{attribute 'enable_dynamic_creation'}
FUNCTION_BLOCK Line EXTENDS Object IMPLEMENTS ILine
VAR_INPUT
END_VAR
VAR_OUTPUT
END_VAR
VAR
	content :STRING(255);
	number :LREAL;
END_VAR

(*

short summary
=================
This abstract property returns the class name of the concrete object, 
which is useful for logging/debugging purpose or to check the class name
for ``__DELETE`` in factories (sometimes it's necessary to do more 
than just to free the memory).

.. <legal notes>

legal notes
=================
| SPDX-FileCopyrightText: © 2022 ekvip automation GmbH <info@ekvip.de>
| SPDX-License-Identifier: Apache-2.0
| For details check: Apache-2.0_

.. _Apache-2.0: https://www.apache.org/licenses/LICENSE-2.0

.. </legal notes>

*)
PROPERTY className : CNM_AbstractObject.ClassName
GET
END_GET
END_PROPERTY

METHOD splitBy :IStringContainerList
VAR_INPUT
	splitter	: STRING(255);
	addEmptyEntries :BOOL := FALSE;
END_VAR
VAR
	pContainterList :POINTER TO StringContainerList;
	
	index :INT;
	searchindex :INT;
	textSize :INT;
	splitterSize :INT;
	lastSplit :INT;
	startSearchIndex : UDINT;
	pContainer :POINTER TO Line;
	currentText : STRING(255);
END_VAR
splitterSize := Tc2_Standard.LEN(splitter);
textSize := Tc2_Standard.LEN(THIS^.text);

pContainterList := __NEW(StringContainerList());
splitBy := pContainterList^;

RETURN (splitterSize = 0);

lastSplit := 0;
FOR index := 0 TO textSize DO
	startSearchIndex := index;
	searchindex := 0;
	WHILE(startSearchIndex+searchindex < textSize AND_THEN THIS^.content[startSearchIndex+searchindex] = splitter[searchindex])DO
		IF(searchindex = splitterSize)THEN //10 is newLine $N
			Tc2_System.MEMSET(ADR(currentText), 0, SIZEOF(currentText));
			Tc2_System.MEMCPY(ADR(currentText), ADR(THIS^.content)+startSearchIndex+searchindex, startSearchIndex + searchindex - splitterSize);
			IF(Tc2_Standard.LEN(currentText) = 0 AND NOT addEmptyEntries)THEN
				index := index + searchindex;
				EXIT;
			END_IF
			pContainer := __NEW(Line());
			pContainer^.text := currentText;
			splitBy.append(pContainer^);
			index := index + searchindex;
			lastSplit := index;
			EXIT;
		END_IF
		searchindex := searchindex+1;
	END_WHILE
END_FOR

Tc2_System.MEMSET(ADR(currentText), 0, SIZEOF(currentText));
Tc2_System.MEMCPY(ADR(currentText), ADR(THIS^.content) + lastSplit, index - lastSplit);
IF(Tc2_Standard.LEN(currentText) = 0 AND NOT addEmptyEntries)THEN
	RETURN;
END_IF
pContainer := __NEW(Line());
pContainer^.text := currentText;
splitBy.append(pContainer^);
END_METHOD

PROPERTY text : STRING(255)
GET
text := THIS^.content;
END_GET
SET
THIS^.content := text;
END_SET
END_PROPERTY

PROPERTY value : LREAL
GET
value := THIS^.number;
END_GET
SET
THIS^.number := value;
END_SET
END_PROPERTY

END_FUNCTION_BLOCK

(* stored: Version 1.1.0.1
   POU Line: Id {7b6e3f51-79c2-4027-9e12-15f5f4e60ad8}, SpecialFunc None
   Property className: Id {f17ccc49-279b-4c5b-9cea-b224d7deceb7}
   Get Get: Id {00ad9ba0-6c99-4050-a76f-b21a2decc352}
   Method splitBy: Id {8d60f00c-e4f1-43f8-9091-369ad2f7612c}
   Property text: Id {79dac07b-3bdd-45ae-af6f-81d7a2721ad2}
   Get Get: Id {6fd401ff-7629-4074-a65e-624c5bfa03e0}
   Set Set: Id {dee87da9-a613-4c6c-9d67-42b6fd814ce1}
   Property value: Id {7ee6d61b-e2c5-4f24-b999-2dba45460860}
   Get Get: Id {6e4fb4bf-58bb-45ce-a18a-f45bc2f5c248}
   Set Set: Id {06d6946e-370f-43c4-bbdb-87cf1e0242e8} *)
